{attribute 'linkalways'} 
{attribute 'no_explicit_call' := 'This FB is a CLASS and must be accessed using methods or properties'}
{attribute 'enable_dynamic_creation'}
FUNCTION_BLOCK FINAL EQ_INT EXTENDS Node
VAR
	in1 : _INT(0);
	in2 : _INT(0);
	out : _BOOL(FALSE);
END_VAR

METHOD PUBLIC Clone : I_Node
VAR
	pNode : POINTER TO EQ_INT;
END_VAR
pNode := __NEW(EQ_INT);
Clone := pNode^;
END_METHOD

METHOD FB_init : BOOL
VAR_INPUT
	bInitRetains : BOOL; // if TRUE, the retain variables are initialized (warm start / cold start)
	bInCopyCode : BOOL;  // if TRUE, the instance afterwards gets moved into the copy code (online change)
END_VAR
AddInput('in1',THIS^.in1);
AddInput('in2',THIS^.in2);
AddOutput('out', THIS^.out);
END_METHOD

METHOD PROTECTED OnExecute
VAR
END_VAR
out.Value := in1.Value = in2.Value;
END_METHOD

END_FUNCTION_BLOCK

(* stored: Version 1.1.0.1, ProductVersion 3.1.4024.15
   POU EQ_INT: Id {f29c524f-1646-4e0e-a4bd-48f0bf6f555f}, SpecialFunc None
   Folder Constructor: Id {6510ebec-1bba-4293-ae79-7d19a1f921f9}
   Method Clone: Id {1ee2d6d3-7999-4644-b288-08a22dd091ee}
   Method FB_init: Id {be2dca57-d535-4f41-bfad-bbc03ed9c8f5}
   Method OnExecute: Id {236bc866-1a30-412f-82a8-76f6c1bd84b6} *)
